// TwinCAT 3 PLC project Test_Proj
// ProgramVersion: 3.1.4026.25
// libraries:
//   Tc2_Standard, * (Beckhoff Automation GmbH)
//   Tc2_System, * (Beckhoff Automation GmbH)
//   Tc3_PlcTestSuite, * (Simmel)
//   [Base Library], * (Beckhoff UK)
// project tree:
//   Mocks/ MockLogger.TcPOU, MockObject.TcPOU, MockCyclic.TcPOU, MockInit.TcPOU, MockAbortable.TcPOU, MockResettable.TcPOU
//   / PlcTask.TcTTO
//   POUs/ MAIN.TcPOU, ObjectTestSuite.TcPOU, RunnerTestSuite.TcPOU, TraceTestSuite.TcPOU
// real-time tasks:
//   TASK PlcTask: cycle T#10ms, priority 20, ADS port 350

CONFIGURATION Test_Proj
    RESOURCE PLC ON TwinCAT3
        TASK PlcTask(INTERVAL := T#10ms, PRIORITY := 20);
        PROGRAM MAIN WITH PlcTask : MAIN;
    END_RESOURCE
END_CONFIGURATION

// ---- POUs/MAIN.TcPOU
PROGRAM MAIN
VAR
	RunnerTests : RunnerTestSuite;
	ObjectTests : ObjectTestSuite;
	TraceTests : TraceTestSuite;
END_VAR

RunnerTests();
ObjectTests();
TraceTests();

END_PROGRAM

// ---- POUs/RunnerTestSuite.TcPOU
FUNCTION_BLOCK RunnerTestSuite
VAR
	ReRun : BOOL;
	RunnerTestSuite : TestSuite<TestSuiteParameter.MaxTestCount>(ResultFile := JUnitResultFile) := (TestSuiteName := 'Runner Test Suite');
END_VAR

ConfirmInitModulesComplete_Test();
ConfirmRunnerCanDeregAllModules_Test();
IncrementAbortCountWhenAdded_Test();
IncrementCyclicCountWhenAdded_Test();
IncrementInitObjCountWhenAdded_Test();
IncrementObjectCountWhenAdded_Test();
IncrementResetCountWhenAdded_Test();
RejectAddingNullAbort_Test();
RejectAddingNullCyclic_Test();
RejectAddingNullInit_Test();
RejectAddingNullObj_Test();
RejectAddingNullReset_Test();
RejectAddingSameAbort_Test();
RejectAddingSameCyclic_Test();
RejectAddingSameInit_Test();
RejectAddingSameObj_Test();
RejectAddingSameReset_Test();
RejectAddingTooManyAbort_Test();
RejectAddingTooManyCyclic_Test();
RejectAddingTooManyInit_Test();
RejectAddingTooManyObj_Test();
RejectAddingTooManyReset_Test();
RejectInitCallWithNoModules_Test();
RejectInvalidInterface_Test();
RunnerAcceptsModule_Test();
IF ReRun THEN
	TestSuite.ReRunTests();
	ReRun := FALSE;
END_IF

METHOD ConfirmInitModulesComplete_Test : BOOL
VAR_INST
	Expected : BOOL;
	Actual	 : BOOL;
END_VAR
VAR
	TestRunner : ObjectRunner<99>;
	TestMockObj : MockInit(Name := 'MockInit');
END_VAR
IF RunnerTestSuite.Test(__POUNAME()).ExecuteTest() THEN
	Expected := TRUE;
	TestRunner.Register(TestMockObj);
	IF Succeeded(TestRunner.Initialise()) THEN
		Actual := TestRunner.InitialisationComplete;
		TestRunner.DeregisterAll();
		RunnerTestSuite.Test(__POUNAME()).AssertEqual(Expected, Actual);
	END_IF
END_IF
END_METHOD

METHOD ConfirmRunnerCanDeregAllModules_Test : BOOL
VAR_INST
	Expected : INT;
	Actual	 : INT;
END_VAR
VAR
	TestRunner : ObjectRunner<99>;
	TestMockObj1 : MockObject(Name := 'MockObj1');
	TestMockObj2 : MockObject(Name := 'MockObj2');
END_VAR
IF RunnerTestSuite.Test(__POUNAME()).ExecuteTest() THEN
	Expected := 0;
	TestRunner.Register(TestMockObj1);
	TestRunner.Register(TestMockObj2);
	Actual := TestRunner.RegisteredObjectCount;
	TestRunner.DeregisterAll();
	Actual := TestRunner.RegisteredObjectCount;
	RunnerTestSuite.Test(__POUNAME()).AssertEqual(Expected, Actual);
END_IF
END_METHOD

METHOD IncrementAbortCountWhenAdded_Test : BOOL
VAR_INST
	Expected : INT := 1;
	Actual	 : INT;
END_VAR
VAR
	TestRunner : ObjectRunner<99>;
	TestMockObj : MockAbortable(Name := 'MockReset');
END_VAR
IF RunnerTestSuite.Test(__POUNAME()).ExecuteTest() THEN
	TestRunner.RegisterAbortable(TestMockObj);
	Actual := TestRunner.AbortableModuleCount;
	RunnerTestSuite.Test(__POUNAME()).AssertEqual(Expected, Actual);
	TestRunner.DeregisterAll();
END_IF
END_METHOD

METHOD IncrementCyclicCountWhenAdded_Test : BOOL
VAR_INST
	Expected : INT := 1;
	Actual	 : INT;
END_VAR
VAR
	TestRunner : ObjectRunner<99>;
	TestMockObj : MockCyclic(Name := 'MockCyclic');
END_VAR
IF RunnerTestSuite.Test(__POUNAME()).ExecuteTest() THEN
	TestRunner.RegisterCyclic(TestMockObj);
	Actual := TestRunner.CyclicModuleCount;
	RunnerTestSuite.Test(__POUNAME()).AssertEqual(Expected, Actual);
	TestRunner.DeregisterAll();
END_IF
END_METHOD

METHOD IncrementInitObjCountWhenAdded_Test : BOOL
VAR_INST
	Expected : INT := 1;
	Actual	 : INT;
END_VAR
VAR
	TestRunner : ObjectRunner<99>;
	TestMockObj : MockInit(Name := 'MockInit');
END_VAR
IF RunnerTestSuite.Test(__POUNAME()).ExecuteTest() THEN
	TestRunner.RegisterInitialisable(TestMockObj);
	Actual := TestRunner.InitialisableModuleCount;
	RunnerTestSuite.Test(__POUNAME()).AssertEqual(Expected, Actual);
	TestRunner.DeregisterAll();
END_IF
END_METHOD

METHOD IncrementObjectCountWhenAdded_Test : BOOL
VAR_INST
	Expected : INT := 1;
	Actual	 : INT;
END_VAR
VAR
	TestRunner : ObjectRunner<99>;
	TestMockObj : MockObject(Name := 'MockObj');
END_VAR
IF RunnerTestSuite.Test(__POUNAME()).ExecuteTest() THEN
	TestRunner.RegisterObject(TestMockObj);
	Actual := TestRunner.RegisteredObjectCount;
	RunnerTestSuite.Test(__POUNAME()).AssertEqual(Expected, Actual);
	TestRunner.DeregisterAll();
END_IF
END_METHOD

METHOD IncrementResetCountWhenAdded_Test : BOOL
VAR_INST
	Expected : INT := 1;
	Actual	 : INT;
END_VAR
VAR
	TestRunner : ObjectRunner<99>;
	TestMockObj : MockResettable(Name := 'MockReset');
END_VAR
IF RunnerTestSuite.Test(__POUNAME()).ExecuteTest() THEN
	TestRunner.RegisterResettable(TestMockObj);
	Actual := TestRunner.ResettableModuleCount;
	RunnerTestSuite.Test(__POUNAME()).AssertEqual(Expected, Actual);
	TestRunner.DeregisterAll();
END_IF
END_METHOD

METHOD RejectAddingNullAbort_Test : BOOL
VAR_INST
	Expected : HRESULT := -1;
	Actual	 : HRESULT;
END_VAR
VAR
	TestRunner : ObjectRunner<99>;
END_VAR
IF RunnerTestSuite.Test(__POUNAME()).ExecuteTest() THEN
	Actual :=  TestRunner.RegisterAbortable(16#00);
	RunnerTestSuite.Test(__POUNAME()).AssertEqual(Expected, Actual);
	TestRunner.DeregisterAll();
END_IF
END_METHOD

METHOD RejectAddingNullCyclic_Test : BOOL
VAR_INST
	Expected : HRESULT := -1;
	Actual	 : HRESULT;
END_VAR
VAR
	TestRunner : ObjectRunner<99>;
END_VAR
IF RunnerTestSuite.Test(__POUNAME()).ExecuteTest() THEN
	Actual :=  TestRunner.RegisterCyclic(16#00);
	RunnerTestSuite.Test(__POUNAME()).AssertEqual(Expected, Actual);
	TestRunner.DeregisterAll();
END_IF
END_METHOD

METHOD RejectAddingNullInit_Test : BOOL
VAR_INST
	Expected : HRESULT := -1;
	Actual	 : HRESULT;
END_VAR
VAR
	TestRunner : ObjectRunner<99>;
END_VAR
IF RunnerTestSuite.Test(__POUNAME()).ExecuteTest() THEN
	Actual :=  TestRunner.RegisterInitialisable(16#00);
	RunnerTestSuite.Test(__POUNAME()).AssertEqual(Expected, Actual);
	TestRunner.DeregisterAll();
END_IF
END_METHOD

METHOD RejectAddingNullObj_Test : BOOL
VAR_INST
	Expected : HRESULT := -1;
	Actual	 : HRESULT;
END_VAR
VAR
	TestRunner : ObjectRunner<99>;
END_VAR
IF RunnerTestSuite.Test(__POUNAME()).ExecuteTest() THEN
	Actual :=  TestRunner.RegisterObject(16#00);
	RunnerTestSuite.Test(__POUNAME()).AssertEqual(Expected, Actual);
	TestRunner.DeregisterAll();
END_IF
END_METHOD

METHOD RejectAddingNullReset_Test : BOOL
VAR_INST
	Expected : HRESULT := -1;
	Actual	 : HRESULT;
END_VAR
VAR
	TestRunner : ObjectRunner<99>;
END_VAR
IF RunnerTestSuite.Test(__POUNAME()).ExecuteTest() THEN
	Actual :=  TestRunner.RegisterResettable(16#00);
	RunnerTestSuite.Test(__POUNAME()).AssertEqual(Expected, Actual);
	TestRunner.DeregisterAll();
END_IF
END_METHOD

METHOD RejectAddingSameAbort_Test : BOOL
VAR_INST
	Expected : HRESULT := -3;
	Actual	 : HRESULT;
END_VAR
VAR
	TestRunner : ObjectRunner<99>;
	TestMockObj : MockAbortable(Name := 'MockAbort');
END_VAR
IF RunnerTestSuite.Test(__POUNAME()).ExecuteTest() THEN
	TestRunner.RegisterAbortable(TestMockObj);
	Actual :=  TestRunner.RegisterAbortable(TestMockObj);
	RunnerTestSuite.Test(__POUNAME()).AssertEqual(Expected, Actual);
	TestRunner.DeregisterAll();
END_IF
END_METHOD

METHOD RejectAddingSameCyclic_Test : BOOL
VAR_INST
	Expected : HRESULT := -3;
	Actual	 : HRESULT;
END_VAR
VAR
	TestRunner : ObjectRunner<99>;
	TestMockObj : MockCyclic(Name := 'Mockcyclic');
END_VAR
IF RunnerTestSuite.Test(__POUNAME()).ExecuteTest() THEN
	TestRunner.RegisterCyclic(TestMockObj);
	Actual := TestRunner.RegisterCyclic(TestMockObj);
	RunnerTestSuite.Test(__POUNAME()).AssertEqual(Expected, Actual);
	TestRunner.DeregisterAll();
END_IF
END_METHOD

METHOD RejectAddingSameInit_Test : BOOL
VAR_INST
	Expected : HRESULT := -3;
	Actual	 : HRESULT;
END_VAR
VAR
	TestRunner : ObjectRunner<99>;
	TestMockObj : MockInit(Name := 'MockInit');
END_VAR
IF RunnerTestSuite.Test(__POUNAME()).ExecuteTest() THEN
	TestRunner.RegisterInitialisable(TestMockObj);
	Actual := TestRunner.RegisterInitialisable(TestMockObj);
	RunnerTestSuite.Test(__POUNAME()).AssertEqual(Expected, Actual);
	TestRunner.DeregisterAll();
END_IF
END_METHOD

METHOD RejectAddingSameObj_Test : BOOL
VAR_INST
	Expected : HRESULT := -3;
	Actual	 : HRESULT;
END_VAR
VAR
	TestRunner : ObjectRunner<99>;
	TestMockObj : MockObject(Name := 'MockObj');
END_VAR
IF RunnerTestSuite.Test(__POUNAME()).ExecuteTest() THEN
	TestRunner.RegisterObject(TestMockObj);
	Actual := TestRunner.RegisterObject(TestMockObj);
	RunnerTestSuite.Test(__POUNAME()).AssertEqual(Expected, Actual);
	TestRunner.DeregisterAll();
END_IF
END_METHOD

METHOD RejectAddingSameReset_Test : BOOL
VAR_INST
	Expected : HRESULT := -3;
	Actual	 : HRESULT;
END_VAR
VAR
	TestRunner : ObjectRunner<99>;
	TestMockObj : MockResettable(Name := 'MockReset');
END_VAR
IF RunnerTestSuite.Test(__POUNAME()).ExecuteTest() THEN
	TestRunner.RegisterResettable(TestMockObj);
	Actual := TestRunner.RegisterResettable(TestMockObj);
	RunnerTestSuite.Test(__POUNAME()).AssertEqual(Expected, Actual);
	TestRunner.DeregisterAll();
END_IF
END_METHOD

METHOD RejectAddingTooManyAbort_Test : BOOL
VAR_INST
	Expected : HRESULT := -2;
	Actual	 : HRESULT;
END_VAR
VAR
	TestRunner : ObjectRunner<1>;
	TestMockObj : MockAbortable(Name := 'MockAbort');
END_VAR
IF RunnerTestSuite.Test(__POUNAME()).ExecuteTest() THEN
	TestRunner.RegisterAbortable(TestMockObj);
	Actual := TestRunner.RegisterAbortable(TestMockObj);
	RunnerTestSuite.Test(__POUNAME()).AssertEqual(Expected, Actual);
	TestRunner.DeregisterAll();
END_IF
END_METHOD

METHOD RejectAddingTooManyCyclic_Test : BOOL
VAR_INST
	Expected : HRESULT := -2;
	Actual	 : HRESULT;
END_VAR
VAR
	TestRunner : ObjectRunner<1>;
	TestMockObj : MockCyclic(Name := 'MockCyclic');
END_VAR
IF RunnerTestSuite.Test(__POUNAME()).ExecuteTest() THEN
	TestRunner.RegisterCyclic(TestMockObj);
	Actual := TestRunner.RegisterCyclic(TestMockObj);
	RunnerTestSuite.Test(__POUNAME()).AssertEqual(Expected, Actual);
	TestRunner.DeregisterAll();
END_IF
END_METHOD

METHOD RejectAddingTooManyInit_Test : BOOL
VAR_INST
	Expected : HRESULT := -2;
	Actual	 : HRESULT;
END_VAR
VAR
	TestRunner : ObjectRunner<1>;
	TestMockObj : MockInit(Name := 'MockInit');
END_VAR
IF RunnerTestSuite.Test(__POUNAME()).ExecuteTest() THEN
	TestRunner.RegisterInitialisable(TestMockObj);
	Actual := TestRunner.RegisterInitialisable(TestMockObj);
	RunnerTestSuite.Test(__POUNAME()).AssertEqual(Expected, Actual);
	TestRunner.DeregisterAll();
END_IF
END_METHOD

METHOD RejectAddingTooManyObj_Test : BOOL
VAR_INST
	Expected : HRESULT := -2;
	Actual	 : HRESULT;
END_VAR
VAR
	TestRunner : ObjectRunner<1>;
	TestMockObj : MockObject(Name := 'MockObj');
END_VAR
IF RunnerTestSuite.Test(__POUNAME()).ExecuteTest() THEN
	TestRunner.RegisterObject(TestMockObj);
	Actual := TestRunner.RegisterObject(TestMockObj);
	RunnerTestSuite.Test(__POUNAME()).AssertEqual(Expected, Actual);
	TestRunner.DeregisterAll();
END_IF
END_METHOD

METHOD RejectAddingTooManyReset_Test : BOOL
VAR_INST
	Expected : HRESULT := -2;
	Actual	 : HRESULT;
END_VAR
VAR
	TestRunner : ObjectRunner<1>;
	TestMockObj : MockResettable(Name := 'MockReset');
END_VAR
IF RunnerTestSuite.Test(__POUNAME()).ExecuteTest() THEN
	TestRunner.RegisterResettable(TestMockObj);
	Actual := TestRunner.RegisterResettable(TestMockObj);
	RunnerTestSuite.Test(__POUNAME()).AssertEqual(Expected, Actual);
	TestRunner.DeregisterAll();
END_IF
END_METHOD

METHOD RejectInitCallWithNoModules_Test : BOOL
VAR_INST
	Expected : BOOL := TRUE;
	Actual	 : BOOL;
END_VAR
VAR
	TestRunner : ObjectRunner<99>;
END_VAR
IF RunnerTestSuite.Test(__POUNAME()).ExecuteTest() THEN
	TestRunner.Initialise();
	Actual := TestRunner.InitialisationComplete;
	RunnerTestSuite.Test(__POUNAME()).AssertEqual(Expected, Actual);
	TestRunner.DeregisterAll();
END_IF
END_METHOD

METHOD RejectInvalidInterface_Test : BOOL
VAR_INST
	Expected : HRESULT := -1;
	Actual	 : HRESULT;
END_VAR
VAR
	TestRunner : ObjectRunner<99>;
END_VAR
IF RunnerTestSuite.Test(__POUNAME()).ExecuteTest() THEN
	Actual := TestRunner.Register(16#0);
	RunnerTestSuite.Test(__POUNAME()).AssertEqual(Expected, Actual);
END_IF
END_METHOD

METHOD RunnerAcceptsModule_Test : BOOL
VAR_INST
	Expected : BOOL := TRUE;
	Actual	 : BOOL;
END_VAR
VAR
	TestRunner : ObjectRunner<99>;
	TestMockObj : MockObject(Name := 'MockObj');
END_VAR
IF RunnerTestSuite.Test(__POUNAME()).ExecuteTest() THEN
	Actual := SuCCEEDED(TestRunner.Register(TestMockObj));
	RunnerTestSuite.Test(__POUNAME()).AssertEqual(Expected, Actual);
	TestRunner.DeregisterAll();
END_IF
END_METHOD

END_FUNCTION_BLOCK

// ---- Mocks/MockInit.TcPOU
FUNCTION_BLOCK MockInit EXTENDS Object IMPLEMENTS I_Initialisable
VAR
	_isRegistered : BOOL;
END_VAR

METHOD Initialise : HRESULT
END_METHOD

{warning 'Add property implementation'}
PROPERTY Initialised : BOOL
GET
Initialised := TRUE;
END_GET
END_PROPERTY

METHOD IsRegistered : BOOL
VAR_INPUT
END_VAR
IsRegistered := _isRegistered;
END_METHOD

METHOD RegisterWithParent
VAR_INPUT
	Parent	: I_HostObjects;
END_VAR
IF NOT _isRegistered THEN
	IF SUCCEEDED(Parent.RegisterInitialisable(THIS^)) THEN
		_isRegistered := TRUE;
	ELSE
		_isRegistered := FALSE;
	END_IF
END_IF
END_METHOD

END_FUNCTION_BLOCK

// ---- Mocks/MockObject.TcPOU
FUNCTION_BLOCK MockObject EXTENDS Object
VAR
	_isRegistered : BOOL;
END_VAR

METHOD IsRegistered : BOOL
VAR_INPUT
END_VAR
IsRegistered := _isRegistered;
END_METHOD

METHOD RegisterWithParent
VAR_INPUT
	Parent	: I_HostObjects;
END_VAR
IF NOT _isRegistered THEN
	IF SUCCEEDED(Parent.RegisterObject(THIS^)) THEN
		_isRegistered := TRUE;
	ELSE
		_isRegistered := FALSE;
	END_IF
END_IF
END_METHOD

END_FUNCTION_BLOCK

// ---- Mocks/MockAbortable.TcPOU
FUNCTION_BLOCK MockAbortable EXTENDS Object IMPLEMENTS I_Abortable
VAR
	_isRegistered : BOOL;
END_VAR

METHOD Abort : Base_Library.HRESULT
END_METHOD

METHOD IsRegistered : BOOL
VAR_INPUT
END_VAR
IsRegistered := _isRegistered;
END_METHOD

METHOD RegisterWithParent
VAR_INPUT
	Parent	: I_HostObjects;
END_VAR
IF NOT _isRegistered THEN
	IF SUCCEEDED(Parent.RegisterAbortable(THIS^)) THEN
		_isRegistered := TRUE;
	ELSE
		_isRegistered := FALSE;
	END_IF
END_IF
END_METHOD

END_FUNCTION_BLOCK

// ---- Mocks/MockCyclic.TcPOU
FUNCTION_BLOCK MockCyclic EXTENDS CyclicBase
VAR
	_isRegistered : BOOL;
END_VAR

METHOD Cycle : HRESULT
END_METHOD

METHOD IsRegistered : BOOL
VAR_INPUT
END_VAR
IsRegistered := _isRegistered;
END_METHOD

METHOD RegisterWithParent
VAR_INPUT
	Parent	: I_HostObjects;
END_VAR
IF NOT _isRegistered THEN
	IF SUCCEEDED( Parent.RegisterCyclic(THIS^)) THEN
		_isRegistered := TRUE;
	ELSE
		_isRegistered := FALSE;
	END_IF
END_IF
END_METHOD

END_FUNCTION_BLOCK

// ---- Mocks/MockResettable.TcPOU
FUNCTION_BLOCK MockResettable EXTENDS Object IMPLEMENTS I_Resettable
VAR
	_isRegistered : BOOL;
END_VAR

METHOD IsRegistered : BOOL
VAR_INPUT
END_VAR
IsRegistered := _isRegistered;
END_METHOD

METHOD RegisterWithParent
VAR_INPUT
	Parent	: I_HostObjects;
END_VAR
IF NOT _isRegistered THEN
	IF SUCCEEDED( Parent.RegisterResettable(THIS^)) THEN
		_isRegistered := TRUE;
	ELSE
		_isRegistered := FALSE;
	END_IF
END_IF
END_METHOD

METHOD Reset : Base_Library.HRESULT
END_METHOD

END_FUNCTION_BLOCK

// ---- POUs/ObjectTestSuite.TcPOU
FUNCTION_BLOCK ObjectTestSuite
VAR
	ReRun : BOOL;
	ObjTestSuite : TestSuite<TestSuiteParameter.MaxTestCount>(ResultFile := JUnitResultFile) := (TestSuiteName := 'Object Test Suite');
END_VAR

ObjectAcceptsName_Test();
IF ReRun THEN
	ObjTestSuite.ReRunTests();
	ReRun := FALSE;
END_IF

METHOD ObjectAcceptsName_Test
VAR_INST
	Expected : BOOL := TRUE;
	Actual	 : BOOL;
END_VAR
VAR
	TestMockObj : MockObject(Name := 'Bob');
END_VAR
IF ObjTestSuite.Test(__POUNAME()).ExecuteTest() THEN
	Expected := TRUE;
	Actual := TestMockObj.Name = 'Bob';
	ObjTestSuite.Test(__POUNAME()).AssertEqual(Expected, Actual);
END_IF
END_METHOD

END_FUNCTION_BLOCK

// ---- POUs/TraceTestSuite.TcPOU
FUNCTION_BLOCK TraceTestSuite
VAR
	TraceTestSuite : TestSuite<TestSuiteParameter.MaxTestCount>(ResultFile := JUnitResultFile) := (TestSuiteName := 'Runner Test Suite');
END_VAR

SubscribeAddsLogger();
UnsubscribeRemovesLogger();
TraceLevelPropertyReturnsAssignedValue();
VerboseLogsWhenTraceLevelVerbose();
VerboseDoesNotLogAbovelVerbose();
InfoLogsBelowInfoLevel();
InfoDoesNotLogAboebInfoLevel();
WarningLogsBelowWarningLevel();
WarningDoesNotLogAbovebWarningLevel();
ErrorDoesNotLogAboveErrorLevel();
ErrorLogsBelowErrorLevel();
CriticalLogsAtCriticalLevel();
CriticalLogsBelowCriticalLevel();
MessageSentToAllSubscribedLoggers();
InfoForwardsCorrectSeverity();

METHOD CriticalLogsAtCriticalLevel
VAR
	Expected : UINT := 1;
	Actual	 : UINT;
	TestTrace : Trace<1>;
	TestLogger : MockLogger;
END_VAR
IF TraceTestSuite.Test(__POUNAME()).ExecuteTest() THEN
	TestTrace.TraceLevel := TcEventSeverityExt.Critical;
	TestTrace.Subscribe(TestLogger);
	TestTrace.Critical('Source', 'Message');
	Actual := TestLogger.CallCount;
	TraceTestSuite.Test(__POUNAME()).AssertEqual(Expected, Actual);
END_IF
END_METHOD

METHOD CriticalLogsBelowCriticalLevel
VAR
	Expected : UINT := 1;
	Actual	 : UINT;
	TestTrace : Trace<1>;
	TestLogger : MockLogger;
END_VAR
IF TraceTestSuite.Test(__POUNAME()).ExecuteTest() THEN
	TestTrace.TraceLevel := TcEventSeverityExt.verbose;
	TestTrace.Subscribe(TestLogger);
	TestTrace.Critical('Source', 'Message');
	Actual := TestLogger.CallCount;
	TraceTestSuite.Test(__POUNAME()).AssertEqual(Expected, Actual);
END_IF
END_METHOD

METHOD ErrorDoesNotLogAboveErrorLevel
VAR
	Expected : UINT := 0;
	Actual	 : UINT;
	TestTrace : Trace<1>;
	TestLogger : MockLogger;
END_VAR
IF TraceTestSuite.Test(__POUNAME()).ExecuteTest() THEN
	TestTrace.TraceLevel := TcEventSeverityExt.Critical;
	TestTrace.Subscribe(TestLogger);
	TestTrace.Error('Source', 'Message');
	Actual := TestLogger.CallCount;
	TraceTestSuite.Test(__POUNAME()).AssertEqual(Expected, Actual);
END_IF
END_METHOD

METHOD ErrorLogsBelowErrorLevel
VAR
	Expected : UINT := 1;
	Actual	 : UINT;
	TestTrace : Trace<1>;
	TestLogger : MockLogger;
END_VAR
IF TraceTestSuite.Test(__POUNAME()).ExecuteTest() THEN
	TestTrace.TraceLevel := TcEventSeverityExt.verbose;
	TestTrace.Subscribe(TestLogger);
	TestTrace.Error('Source', 'Message');
	Actual := TestLogger.CallCount;
	TraceTestSuite.Test(__POUNAME()).AssertEqual(Expected, Actual);
END_IF
END_METHOD

METHOD InfoDoesNotLogAboebInfoLevel
VAR
	Expected : UINT := 0;
	Actual	 : UINT;
	TestTrace : Trace<1>;
	TestLogger : MockLogger;
END_VAR
IF TraceTestSuite.Test(__POUNAME()).ExecuteTest() THEN
	TestTrace.TraceLevel := TcEventSeverityExt.Warning;
	TestTrace.Subscribe(TestLogger);
	TestTrace.Info('Source', 'Message');
	Actual := TestLogger.CallCount;
	TraceTestSuite.Test(__POUNAME()).AssertEqual(Expected, Actual);
END_IF
END_METHOD

METHOD InfoForwardsCorrectSeverity
VAR
	Expected : UINT := 1;
	Actual	 : UINT;
	TestTrace : Trace<1>;
	TestLogger : MockLogger;
END_VAR
IF TraceTestSuite.Test(__POUNAME()).ExecuteTest() THEN
	TestTrace.TraceLevel := TcEventSeverityExt.Verbose;
	TestTrace.Subscribe(TestLogger);
	TestTrace.Info('TestSource', 'TestMessage');
	Actual := TestLogger.LastSeverity;
	TraceTestSuite.Test(__POUNAME()).AssertEqual(Expected, Actual);
END_IF
END_METHOD

METHOD InfoLogsBelowInfoLevel
VAR
	Expected : UINT := 1;
	Actual	 : UINT;
	TestTrace : Trace<1>;
	TestLogger : MockLogger;
END_VAR
IF TraceTestSuite.Test(__POUNAME()).ExecuteTest() THEN
	TestTrace.TraceLevel := TcEventSeverityExt.verbose;
	TestTrace.Subscribe(TestLogger);
	TestTrace.Info('Source', 'Message');
	Actual := TestLogger.CallCount;
	TraceTestSuite.Test(__POUNAME()).AssertEqual(Expected, Actual);
END_IF
END_METHOD

METHOD MessageSentToAllSubscribedLoggers
VAR
	Expected : HRESULT := 2;
	Actual	 : HRESULT;
	TestTrace : Trace<2>;
	TestLogger1 : MockLogger;
	TestLogger2 : MockLogger;
END_VAR
IF TraceTestSuite.Test(__POUNAME()).ExecuteTest() THEN
	TestTrace.TraceLevel := TcEventSeverityExt.Verbose;
	TestTrace.Subscribe(TestLogger1);
	TestTrace.Subscribe(TestLogger2);
	TestTrace.Info('Source', 'Message');
	Actual := TestLogger1.CallCount + TestLogger2.CallCount;
	TraceTestSuite.Test(__POUNAME()).AssertEqual(Expected, Actual);
END_IF
END_METHOD

METHOD SubscribeAddsLogger
VAR
	Expected : UINT := 1;
	Actual	 : UINT;
	TestTrace : Trace<1>;
	TestLogger : MockLogger;
END_VAR
IF TraceTestSuite.Test(__POUNAME()).ExecuteTest() THEN
	TestTrace.TraceLevel := TcEventSeverityExt.Verbose;
	TestTrace.Subscribe(TestLogger);
	TestTrace.Info('Source', 'Message');
	Actual := TestLogger.CallCount;
	TraceTestSuite.Test(__POUNAME()).AssertEqual(Expected, Actual);
END_IF
END_METHOD

METHOD TraceLevelPropertyReturnsAssignedValue
VAR
	TestTrace : Trace<1>;
	Expected : TcEventSeverityExt := TcEventSeverityExt.Error;
	Actual	 : TcEventSeverityExt;
END_VAR
IF TraceTestSuite.Test(__POUNAME()).ExecuteTest() THEN
	TestTrace.TraceLevel := TcEventSeverityExt.Error;
	Actual := TestTrace.TraceLevel;
	TraceTestSuite.Test(__POUNAME()).AssertEqual(Expected, Actual);
END_IF
END_METHOD

METHOD UnsubscribeRemovesLogger
VAR
	Expected : UINT := 0;
	Actual	 : UINT;
	TestTrace : Trace<1>;
	TestLogger : MockLogger;
END_VAR
IF TraceTestSuite.Test(__POUNAME()).ExecuteTest() THEN
	TestTrace.TraceLevel := TcEventSeverityExt.Verbose;
	TestTrace.Subscribe(TestLogger);
	TestTrace.Unsubscribe(TestLogger);
	TestTrace.Info('Source', 'Message');
	Actual := TestLogger.CallCount;
	TraceTestSuite.Test(__POUNAME()).AssertEqual(Expected, Actual);
END_IF
END_METHOD

METHOD VerboseDoesNotLogAbovelVerbose
VAR
	Expected : UINT := 0;
	Actual	 : UINT;
	TestTrace : Trace<1>;
	TestLogger : MockLogger;
END_VAR
IF TraceTestSuite.Test(__POUNAME()).ExecuteTest() THEN
	TestTrace.TraceLevel := TcEventSeverityExt.Warning;
	TestTrace.Subscribe(TestLogger);
	TestTrace.Verbose('Source', 'Message');
	Actual := TestLogger.CallCount;
	TraceTestSuite.Test(__POUNAME()).AssertEqual(Expected, Actual);
END_IF
END_METHOD

METHOD VerboseLogsWhenTraceLevelVerbose
VAR
	Expected : UINT := 1;
	Actual	 : UINT;
	TestTrace : Trace<1>;
	TestLogger : MockLogger;
END_VAR
IF TraceTestSuite.Test(__POUNAME()).ExecuteTest() THEN
	TestTrace.TraceLevel := TcEventSeverityExt.Verbose;
	TestTrace.Subscribe(TestLogger);
	TestTrace.Verbose('Source', 'Message');
	Actual := TestLogger.CallCount;
	TraceTestSuite.Test(__POUNAME()).AssertEqual(Expected, Actual);
END_IF
END_METHOD

METHOD WarningDoesNotLogAbovebWarningLevel
VAR
	Expected : UINT := 0;
	Actual	 : UINT;
	TestTrace : Trace<1>;
	TestLogger : MockLogger;
END_VAR
IF TraceTestSuite.Test(__POUNAME()).ExecuteTest() THEN
	TestTrace.TraceLevel := TcEventSeverityExt.Critical;
	TestTrace.Subscribe(TestLogger);
	TestTrace.Warning('Source', 'Message');
	Actual := TestLogger.CallCount;
	TraceTestSuite.Test(__POUNAME()).AssertEqual(Expected, Actual);
END_IF
END_METHOD

METHOD WarningLogsBelowWarningLevel
VAR
	Expected : UINT := 1;
	Actual	 : UINT;
	TestTrace : Trace<1>;
	TestLogger : MockLogger;
END_VAR
IF TraceTestSuite.Test(__POUNAME()).ExecuteTest() THEN
	TestTrace.TraceLevel := TcEventSeverityExt.Info;
	TestTrace.Subscribe(TestLogger);
	TestTrace.Warning('Source', 'Message');
	Actual := TestLogger.CallCount;
	TraceTestSuite.Test(__POUNAME()).AssertEqual(Expected, Actual);
END_IF
END_METHOD

END_FUNCTION_BLOCK

// ---- Mocks/MockLogger.TcPOU
FUNCTION_BLOCK MockLogger IMPLEMENTS I_TraceLogger
VAR
	_CallCount : UINT;
	_LastSource : T_MaxString;
	_LastMessage : T_MaxString;
	_LastSeverity : UINT;
END_VAR

PROPERTY CallCount : UINT
GET
CallCount := _CallCount;
END_GET
END_PROPERTY

PROPERTY LastMessage : T_Maxstring
GET
LastMessage := _LastMessage;
END_GET
END_PROPERTY

PROPERTY LastSeverity : UINT
GET
LastSeverity := _LastSeverity;
END_GET
END_PROPERTY

PROPERTY LastSource : T_Maxstring
GET
LastSource := _LastSource;
END_GET
END_PROPERTY

METHOD LogMessage
VAR_INPUT
	Key	: Base_Library.T_MaxString;
	Value	: Base_Library.T_MaxString;
	SourceId	: UDINT := 0;
	TimeStamp	: ULINT := 0;
	MessageId	: UDINT := 1;
	Severity	: USINT := 1;
END_VAR
_CallCount := _CallCount + 1;

_LastSource := key;

_LastMessage := value;

_LastSeverity := Severity;
END_METHOD

END_FUNCTION_BLOCK
